FUNCTION_BLOCK fbSplit
VAR_INPUT
	IN		:REAL;
END_VAR
VAR_OUTPUT
	OUT1	:REAL;
	OUT2	:REAL;
END_VAR
VAR
END_VAR

//Split one input into two outputs
OUT1 := IN;
OUT2 := IN;

END_FUNCTION_BLOCK

(* stored: Version 1.1.0.1, ProductVersion 3.1.4022.6
   POU fbSplit: Id {23601f14-690f-4566-ae73-23eb53cc305b}, SpecialFunc None *)
